PROGRAM MAIN
VAR
	b1: BOOL;
	b2:BOOL;
	c1: BOOL;

END_VAR

b1:=FALSE;
b2:=TRUE;
c1:=FALSE;

END_PROGRAM

(* stored: Version 1.1.0.1, ProductVersion 3.1.4024.11
   POU MAIN: Id {719519df-59da-4ee1-b75d-42692bd0c354}, SpecialFunc None *)
